// Mitsubishi GX Works2 project: data resister with pulse   PLC: FX1N/FX1NC

PROGRAM MAIN
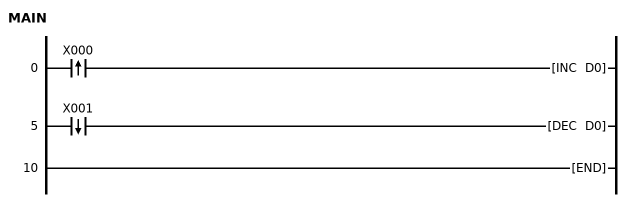
0     LDP     X000
      INC     D0
5     LDF     X001
      DEC     D0
10    END
END_PROGRAM
